Staubli VAL3: CartesianPos.dtx

public pointRx cp = {fatherId=world[0]}
